// TIA Portal V16 export
// export: Created 2023-07-12T06:46:41.6965178Z, ExportSetting WithDefaults, WithReadOnly, DisplayName Totally Integrated Automation Portal, DisplayVersion V16 Update 6, DisplayName TIA Portal Version Control Interface, DisplayVersion V16 Update 2, DisplayName TIA Portal Openness, DisplayVersion V16 Update 6, DisplayName TIA Portal Teamcenter Gateway, DisplayVersion V16, DisplayName SINAMICS Startdrive Advanced, DisplayVersion V16 Update 5, DisplayName SINAMICS Startdrive G130, G150, S120, S150, SINAMICS MV, S210, DisplayVersion V16 Update 5, DisplayName SINAMICS Startdrive G110M, G120, G120C, G120D, G120P, G115D, DisplayVersion V16 Update 5, DisplayName STEP 7 Professional, DisplayVersion V16 Update 6, DisplayName STEP 7 Safety, DisplayVersion V16, DisplayName WinCC Advanced / Unified PC, DisplayVersion V16 Update 6
FUNCTION "FC_Actuators" : Void   // FC13, LAD
{ S7_Optimized_Access := 'TRUE' }
VERSION : 0.1
// stored: AutoNumber true, CodeModifiedDate 2023-07-12T06:46:18.6343226Z, CompileDate 2023-07-12T06:46:27.4474252Z, CreationDate 2023-07-12T06:41:33.7295536Z, HandleErrorsWithinBlock false, InterfaceModifiedDate 2023-06-16T06:31:28.8944821Z, IsConsistent true, IsIECCheckEnabled false, IsKnowHowProtected false, IsWriteProtected false, LibraryConformanceStatus Error: The block contains calls of single instances. Warning: The object contains access to global data blocks. Warning: The block contains direct access to inputs, outputs, bit memories, indirect access to the registry or indirect access to external memory areas that are unknown at the time of compilation. Warning: The object contains access to global PLC constants., ModifiedDate 2023-07-12T06:46:18.6343226Z, ParameterModified 2023-05-11T09:28:46.7777511Z, PLCSimAdvancedSupport true, SetENOAutomatically false, StructureModified 2023-05-11T09:28:46.7777511Z, UDAEnableTagReadback false
   VAR_TEMP
      Safety : Struct
         Estop : Bool;
         Curtain : Bool;
         Proces : Bool;
      END_STRUCT;
      Auto : Bool;
      Actuator : Int;
      AssocValues : Array[1..8] of UInt;
      i : Int;
   END_VAR
BEGIN

REGION Network 1: --------------------------- Movements -----------------------------
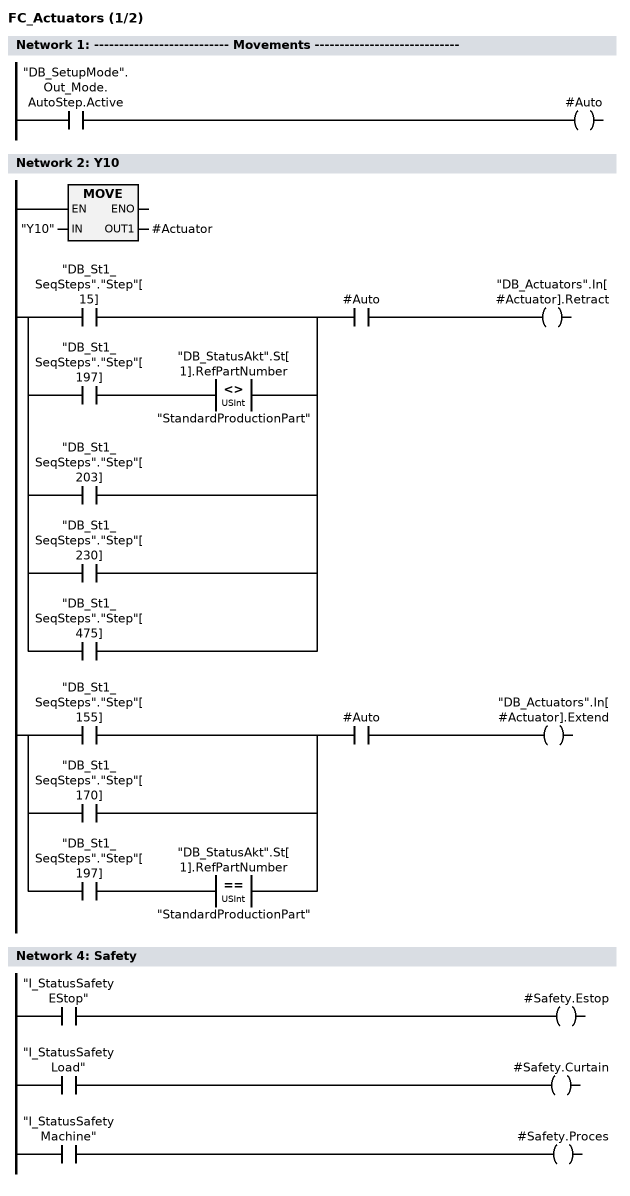
   RUNG wire#powerrail
      Contact( "DB_SetupMode".Out_Mode.AutoStep.Active )
      Coil( #Auto )
   END_RUNG
   // the same network as SCL:
   #Auto := "DB_SetupMode".Out_Mode.AutoStep.Active;
END_REGION

REGION Network 2: Y10
   RUNG wire#powerrail
      Move(in := "Y10", out1 => #Actuator)
   END_RUNG
   RUNG wire#powerrail
      Contact( "DB_St1_SeqSteps"."Step"[15] )
      wire#w1
      Contact( #Auto )
      Coil( "DB_Actuators".In[#Actuator].Retract )
   END_RUNG
   RUNG wire#powerrail
      Contact( "DB_St1_SeqSteps"."Step"[197] )
      { S7_Templates := "SrcType := USInt" } NE_Contact(in1 := "DB_StatusAkt".St[1].RefPartNumber, in2 := "StandardProductionPart")
   END_RUNG wire#w1
   RUNG wire#powerrail
      Contact( "DB_St1_SeqSteps"."Step"[203] )
   END_RUNG wire#w1
   RUNG wire#powerrail
      Contact( "DB_St1_SeqSteps"."Step"[230] )
   END_RUNG wire#w1
   RUNG wire#powerrail
      Contact( "DB_St1_SeqSteps"."Step"[475] )
   END_RUNG wire#w1
   RUNG wire#powerrail
      Contact( "DB_St1_SeqSteps"."Step"[155] )
      wire#w2
      Contact( #Auto )
      Coil( "DB_Actuators".In[#Actuator].Extend )
   END_RUNG
   RUNG wire#powerrail
      Contact( "DB_St1_SeqSteps"."Step"[170] )
   END_RUNG wire#w2
   RUNG wire#powerrail
      Contact( "DB_St1_SeqSteps"."Step"[197] )
      { S7_Templates := "SrcType := USInt" } EQ_Contact(in1 := "DB_StatusAkt".St[1].RefPartNumber, in2 := "StandardProductionPart")
   END_RUNG wire#w2
   // the same network as SCL:
   #Actuator := "Y10";
   "DB_Actuators".In[#Actuator].Retract := ("DB_St1_SeqSteps"."Step"[15] OR ("DB_St1_SeqSteps"."Step"[197] AND ("DB_StatusAkt".St[1].RefPartNumber <> "StandardProductionPart")) OR "DB_St1_SeqSteps"."Step"[203] OR "DB_St1_SeqSteps"."Step"[230] OR "DB_St1_SeqSteps"."Step"[475]) AND #Auto;
   "DB_Actuators".In[#Actuator].Extend := ("DB_St1_SeqSteps"."Step"[155] OR "DB_St1_SeqSteps"."Step"[170] OR ("DB_St1_SeqSteps"."Step"[197] AND ("DB_StatusAkt".St[1].RefPartNumber = "StandardProductionPart"))) AND #Auto;
END_REGION

REGION Network 3: --------------------------- Parameters -----------------------------
END_REGION

REGION Network 4: Safety
   RUNG wire#powerrail
      Contact( "I_StatusSafetyEStop" )
      Coil( #Safety.Estop )
   END_RUNG
   RUNG wire#powerrail
      Contact( "I_StatusSafetyLoad" )
      Coil( #Safety.Curtain )
   END_RUNG
   RUNG wire#powerrail
      Contact( "I_StatusSafetyMachine" )
      Coil( #Safety.Proces )
   END_RUNG
   // the same network as SCL:
   #Safety.Estop := "I_StatusSafetyEStop";
   #Safety.Curtain := "I_StatusSafetyLoad";
   #Safety.Proces := "I_StatusSafetyMachine";
END_REGION

REGION Network 5: Y10
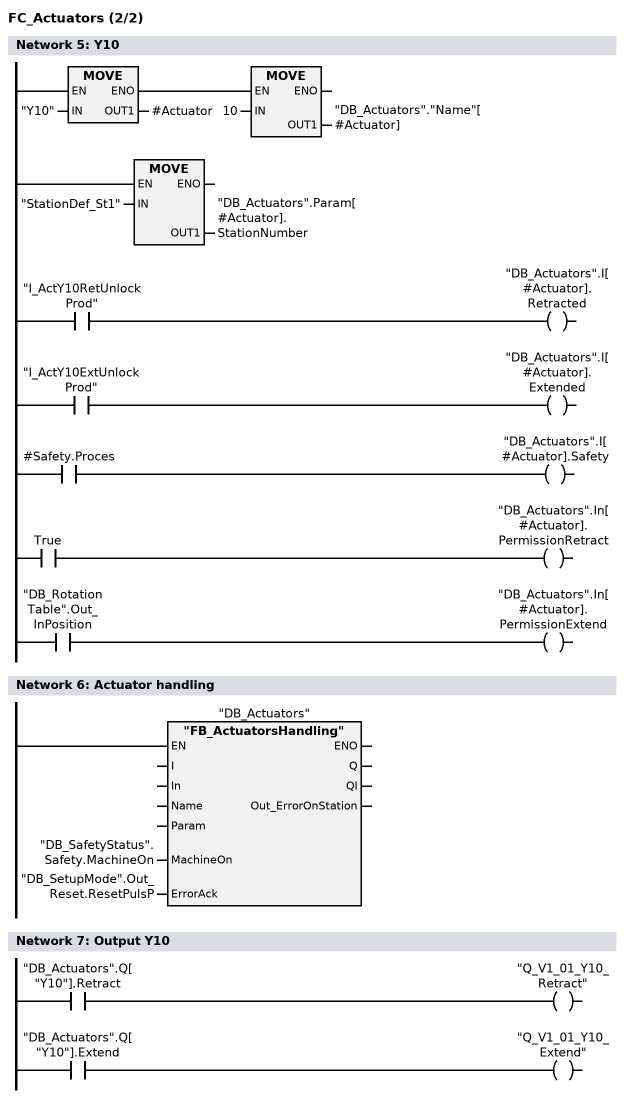
   RUNG wire#powerrail
      Move(in := "Y10", out1 => #Actuator)
      Move(in := 10, out1 => "DB_Actuators"."Name"[#Actuator])
   END_RUNG
   RUNG wire#powerrail
      Move(in := "StationDef_St1", out1 => "DB_Actuators".Param[#Actuator].StationNumber)
   END_RUNG
   RUNG wire#powerrail
      Contact( "I_ActY10RetUnlockProd" )
      Coil( "DB_Actuators".I[#Actuator].Retracted )
   END_RUNG
   RUNG wire#powerrail
      Contact( "I_ActY10ExtUnlockProd" )
      Coil( "DB_Actuators".I[#Actuator].Extended )
   END_RUNG
   RUNG wire#powerrail
      Contact( #Safety.Proces )
      Coil( "DB_Actuators".I[#Actuator].Safety )
   END_RUNG
   RUNG wire#powerrail
      Contact( True )
      Coil( "DB_Actuators".In[#Actuator].PermissionRetract )
   END_RUNG
   RUNG wire#powerrail
      Contact( "DB_RotationTable".Out_InPosition )
      Coil( "DB_Actuators".In[#Actuator].PermissionExtend )
   END_RUNG
   // the same network as SCL:
   #Actuator := "Y10";
   "DB_Actuators"."Name"[#Actuator] := 10;
   "DB_Actuators".Param[#Actuator].StationNumber := "StationDef_St1";
   "DB_Actuators".I[#Actuator].Retracted := "I_ActY10RetUnlockProd";
   "DB_Actuators".I[#Actuator].Extended := "I_ActY10ExtUnlockProd";
   "DB_Actuators".I[#Actuator].Safety := #Safety.Proces;
   "DB_Actuators".In[#Actuator].PermissionRetract := True;
   "DB_Actuators".In[#Actuator].PermissionExtend := "DB_RotationTable".Out_InPosition;
END_REGION

REGION Network 6: Actuator handling
   RUNG wire#powerrail
      "DB_Actuators"(I :=, In :=, "Name" :=, Param :=, MachineOn := "DB_SafetyStatus".Safety.MachineOn, ErrorAck := "DB_SetupMode".Out_Reset.ResetPulsP, Q =>, QI =>, Out_ErrorOnStation =>)
   END_RUNG
   // the same network as SCL:
   "DB_Actuators"(MachineOn := "DB_SafetyStatus".Safety.MachineOn,   // "FB_ActuatorsHandling"
                  ErrorAck := "DB_SetupMode".Out_Reset.ResetPulsP);
END_REGION

REGION Network 7: Output Y10
   RUNG wire#powerrail
      Contact( "DB_Actuators".Q["Y10"].Retract )
      Coil( "Q_V1_01_Y10_Retract" )
   END_RUNG
   RUNG wire#powerrail
      Contact( "DB_Actuators".Q["Y10"].Extend )
      Coil( "Q_V1_01_Y10_Extend" )
   END_RUNG
   // the same network as SCL:
   "Q_V1_01_Y10_Retract" := "DB_Actuators".Q["Y10"].Retract;
   "Q_V1_01_Y10_Extend" := "DB_Actuators".Q["Y10"].Extend;
END_REGION
END_FUNCTION
